INTERFACE I_OpenCommand

PROPERTY IsOpen : Bool
GET
END_GET
END_PROPERTY

METHOD Open
END_METHOD

END_INTERFACE

(* stored: Version 1.1.0.1, ProductVersion 3.1.4024.11
   Itf I_OpenCommand: Id {cae4df8e-f3dc-4178-af73-0811040cc013}
   Property IsOpen: Id {265295e2-ebd9-4fd3-a322-57b798161a3a}
   Get Get: Id {b8a8c704-035e-496b-9550-bc6b814f44b1}
   Method Open: Id {b3a70e25-45f2-42b7-bb12-8db8e9555543} *)
